// TIA Portal V20 export
DATA_BLOCK "ControlNodes"   // DB163
// stored: MemoryReserve 100, Namespace Unit1.Em3
   VAR
      em : "LAF_typeEmControlNode";
      emstate { S7_SetPoint := 'True'} : "LUC_typeStates";
      cm : "Unit1.Em3.typeCmControlNode";
      citiMap : Struct
         PMC : "LER_PMC_Input_Data";
         FlexNet { S7_SetPoint := 'True'} : "LER_FlexNet_Data";
      END_STRUCT;
      topTapeLoading : "Unit1.Em3.typeSequenceControlNode_topTapeLoading";
      topTapeAttachment : "Unit1.Em3.typeSequenceControlNode_topTapeAttachment";
      topTapeFixStage : "Unit1.Em3.typeSequenceControlNode_topTapeFixStage";
      SpecialFunctionMode : Struct
         DryRun : Struct
            JRdetectPV : Array[0..15] of Bool;
         END_STRUCT;
      END_STRUCT;
      cmTopTapeJRDetect : "LBC_typeDigitalSignalControlNode";
      cmTopTapeDiameter : "LBC_typeDigitalSignalControlNode";
      cmTopTapeAxisX : "LBC_typeAxis64PosControlNode";
      cmTopTapeAxisY : "LBC_typeAxis64PosControlNode";
      cmTopTapeLoadingBwdFwd : "LBC_typeTwoWayActuatorControlNode";
      cmTopTapeLoadingClampOpenClose : "LBC_typeTwoWayActuatorControlNode";
      cmTopTapeCutterUpDown : "LBC_typeTwoWayActuatorControlNode";
      cmTopTapeCutterClampUpDown : "LBC_typeTwoWayActuatorControlNode";
      cmTopTapeTensionBwdFwd : "LBC_typeTwoWayActuatorControlNode";
      cmTopTapeAttachmentUpDown : "LBC_typeTwoWayActuatorControlNode";
      cmTopTapeClampTopLeftUpDown : "LBC_typeTwoWayActuatorControlNode";
      cmTopTapeClampTopCenterUpDown : "LBC_typeTwoWayActuatorControlNode";
      cmTopTapeClampTopRightUpDown : "LBC_typeTwoWayActuatorControlNode";
      cmTopTapeClampBtmDownUp : "LBC_typeTwoWayActuatorControlNode";
      cmTopTapeClampAllOpenClose : "LBC_typeTwoWayActuatorControlNode";
      cmTopTapeAttachmentVaccumOffOn : "LBC_typeTwoWayActuatorControlNode";
      cmQrHandyReader : "LER_typeDM8700ControlNode";
   END_VAR
BEGIN
END_DATA_BLOCK
